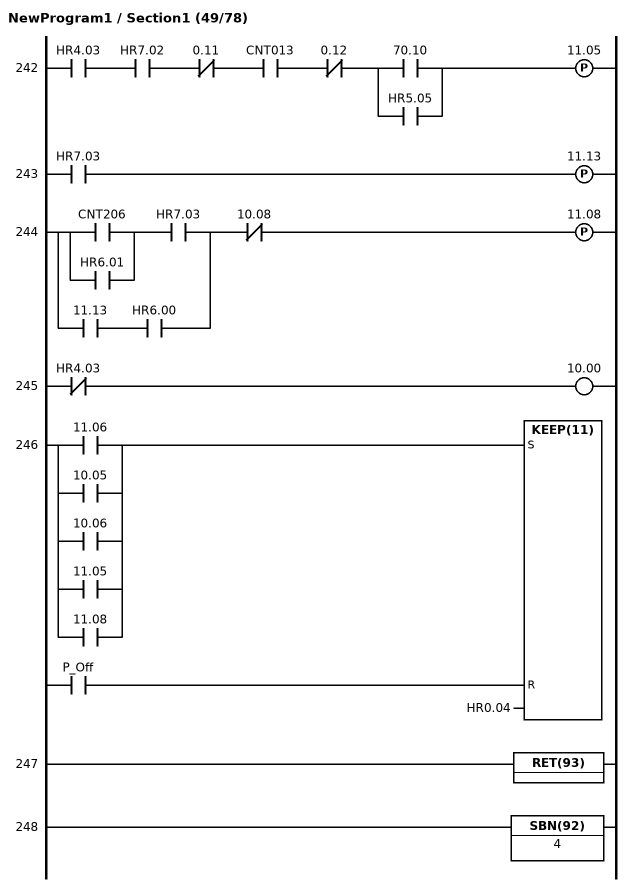
; [picture p48: NewProgram1 / Section1, rungs 242-248]
; rung 242
LD HR4.03
AND HR7.02
ANDNOT 0.11
AND CNT013
ANDNOT 0.12
LD 70.10
OR HR5.05
ANDLD
DIFU(13) 11.05
; rung 243
LD HR7.03
DIFU(13) 11.13
; rung 244
LD CNT206
OR HR6.01
AND HR7.03
LD 11.13
AND HR6.00
ORLD
ANDNOT 10.08
DIFU(13) 11.08
; rung 245
LDNOT HR4.03
OUT 10.00
; rung 246
LD 11.06
OR 10.05
OR 10.06
OR 11.05
OR 11.08
LD P_Off
KEEP(11) HR0.04
; rung 247
RET(93)
; rung 248
SBN(92) 4

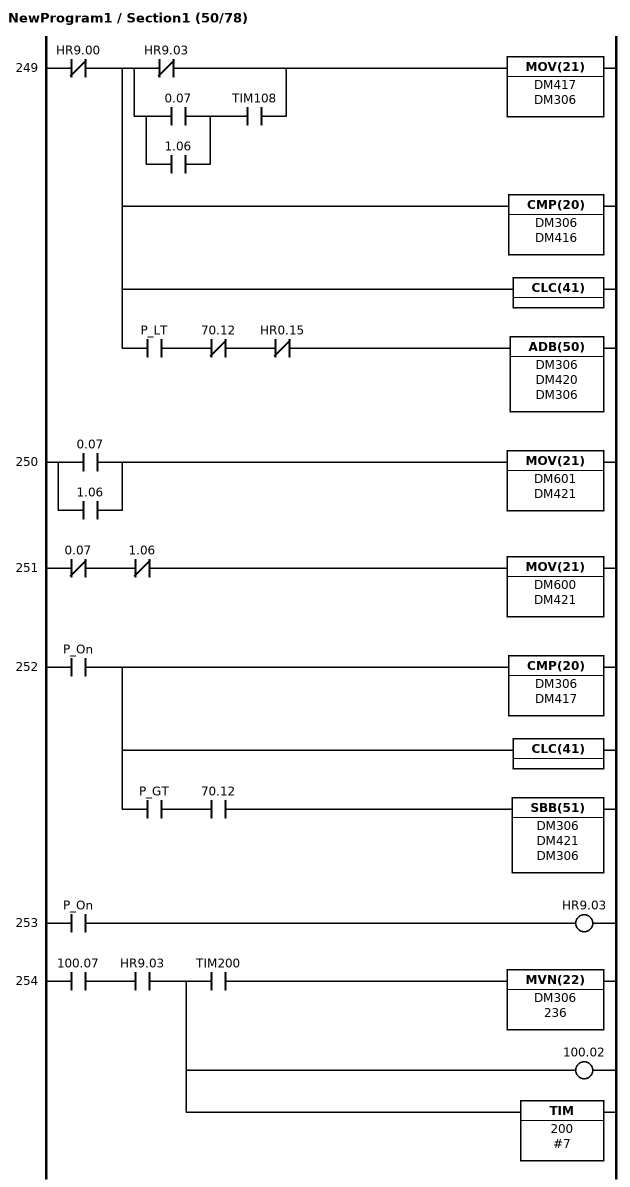
; rung 249
LDNOT HR9.00
OUT TR0
LDNOT HR9.03
LD 0.07
OR 1.06
AND TIM108
ORLD
ANDLD
MOV(21) DM417 DM306
LD TR0
CMP(20) DM306 DM416
CLC(41)
AND P_LT
ANDNOT 70.12
ANDNOT HR0.15
ADB(50) DM306 DM420 DM306
; rung 250
LD 0.07
OR 1.06
MOV(21) DM601 DM421
; rung 251
LDNOT 0.07
ANDNOT 1.06
MOV(21) DM600 DM421
; rung 252
LD P_On
CMP(20) DM306 DM417
CLC(41)
AND P_GT
AND 70.12
SBB(51) DM306 DM421 DM306
; rung 253
LD P_On
OUT HR9.03
; rung 254
LD 100.07
AND HR9.03
OUT TR0
AND TIM200
MVN(22) DM306 236
LD TR0
OUT 100.02
TIM 200 #7

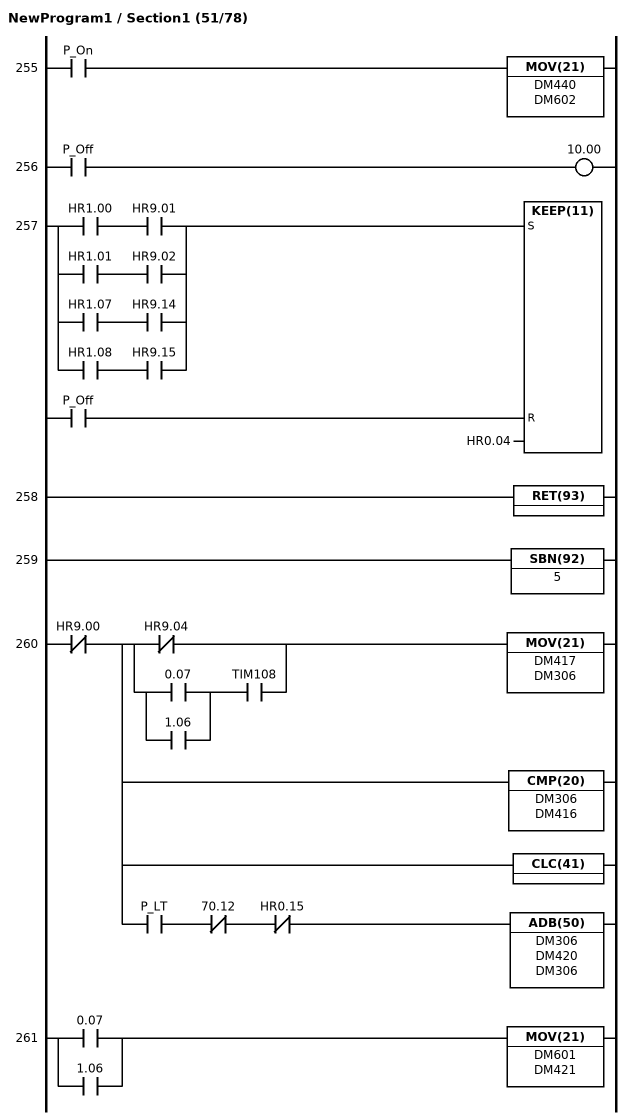
; rung 255
LD P_On
MOV(21) DM440 DM602
; rung 256
LD P_Off
OUT 10.00
; rung 257
LD HR1.00
AND HR9.01
LD HR1.01
AND HR9.02
ORLD
LD HR1.07
AND HR9.14
ORLD
LD HR1.08
AND HR9.15
ORLD
LD P_Off
KEEP(11) HR0.04
; rung 258
RET(93)
; rung 259
SBN(92) 5
; rung 260
LDNOT HR9.00
OUT TR0
LDNOT HR9.04
LD 0.07
OR 1.06
AND TIM108
ORLD
ANDLD
MOV(21) DM417 DM306
LD TR0
CMP(20) DM306 DM416
CLC(41)
AND P_LT
ANDNOT 70.12
ANDNOT HR0.15
ADB(50) DM306 DM420 DM306
; rung 261
LD 0.07
OR 1.06
MOV(21) DM601 DM421

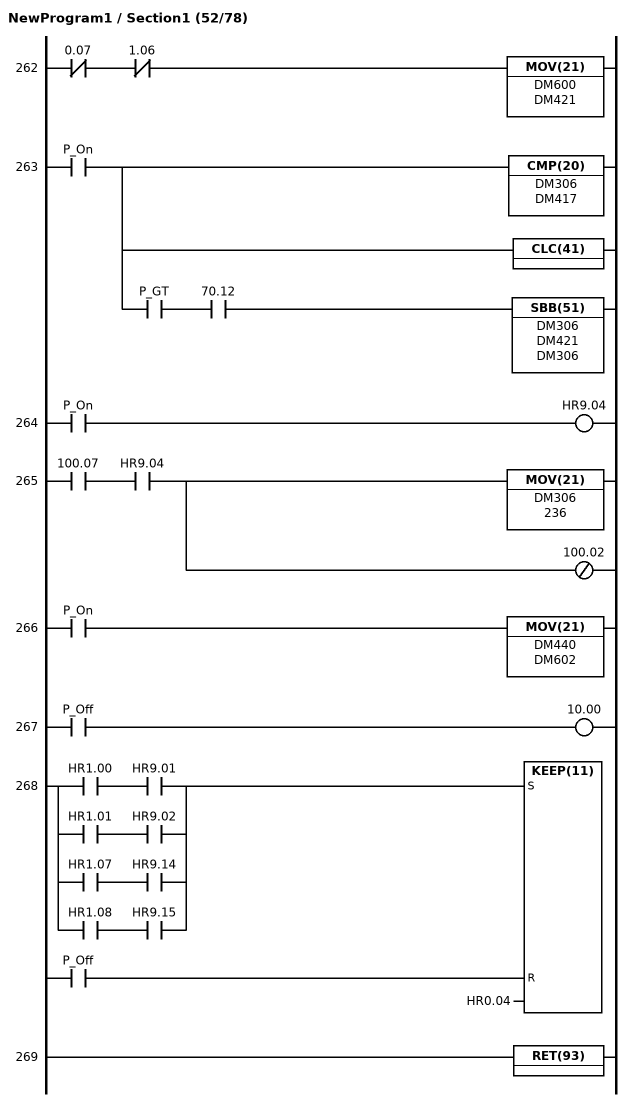
; rung 262
LDNOT 0.07
ANDNOT 1.06
MOV(21) DM600 DM421
; rung 263
LD P_On
CMP(20) DM306 DM417
CLC(41)
AND P_GT
AND 70.12
SBB(51) DM306 DM421 DM306
; rung 264
LD P_On
OUT HR9.04
; rung 265
LD 100.07
AND HR9.04
MOV(21) DM306 236
OUTNOT 100.02
; rung 266
LD P_On
MOV(21) DM440 DM602
; rung 267
LD P_Off
OUT 10.00
; rung 268
LD HR1.00
AND HR9.01
LD HR1.01
AND HR9.02
ORLD
LD HR1.07
AND HR9.14
ORLD
LD HR1.08
AND HR9.15
ORLD
LD P_Off
KEEP(11) HR0.04
; rung 269
RET(93)

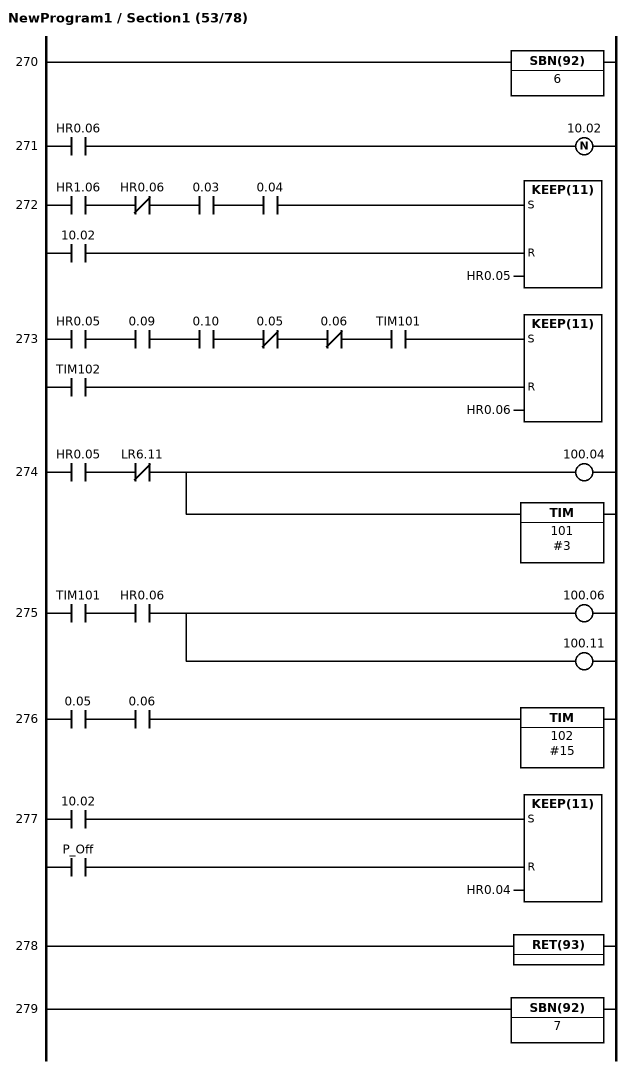
; rung 270
SBN(92) 6
; rung 271
LD HR0.06
DIFD(14) 10.02
; rung 272
LD HR1.06
ANDNOT HR0.06
AND 0.03
AND 0.04
LD 10.02
KEEP(11) HR0.05
; rung 273
LD HR0.05
AND 0.09
AND 0.10
ANDNOT 0.05
ANDNOT 0.06
AND TIM101
LD TIM102
KEEP(11) HR0.06
; rung 274
LD HR0.05
ANDNOT LR6.11
OUT 100.04
TIM 101 #3
; rung 275
LD TIM101
AND HR0.06
OUT 100.06
OUT 100.11
; rung 276
LD 0.05
AND 0.06
TIM 102 #15
; rung 277
LD 10.02
LD P_Off
KEEP(11) HR0.04
; rung 278
RET(93)
; rung 279
SBN(92) 7

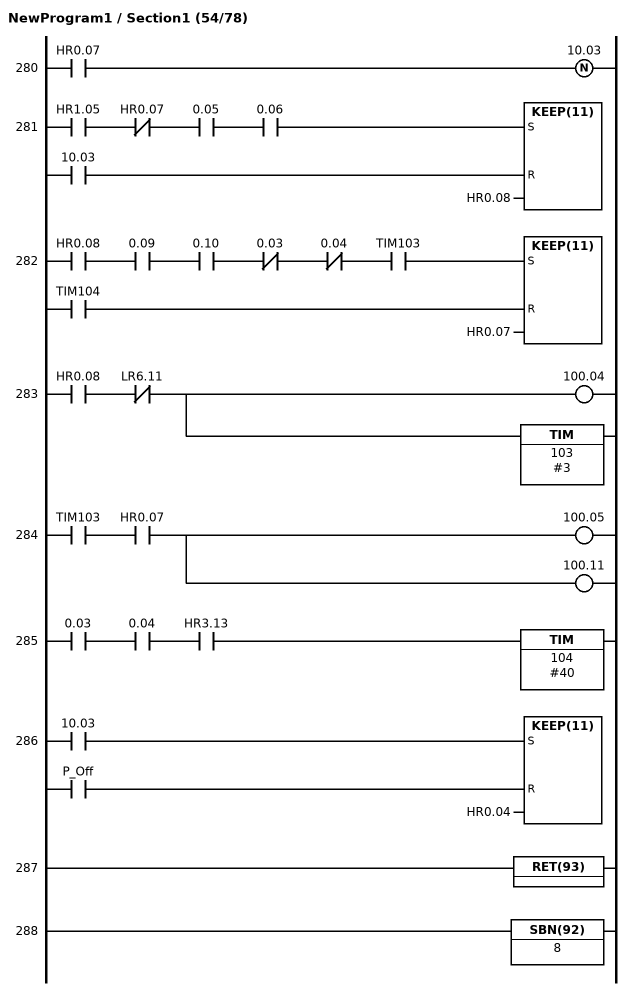
; rung 280
LD HR0.07
DIFD(14) 10.03
; rung 281
LD HR1.05
ANDNOT HR0.07
AND 0.05
AND 0.06
LD 10.03
KEEP(11) HR0.08
; rung 282
LD HR0.08
AND 0.09
AND 0.10
ANDNOT 0.03
ANDNOT 0.04
AND TIM103
LD TIM104
KEEP(11) HR0.07
; rung 283
LD HR0.08
ANDNOT LR6.11
OUT 100.04
TIM 103 #3
; rung 284
LD TIM103
AND HR0.07
OUT 100.05
OUT 100.11
; rung 285
LD 0.03
AND 0.04
AND HR3.13
TIM 104 #40
; rung 286
LD 10.03
LD P_Off
KEEP(11) HR0.04
; rung 287
RET(93)
; rung 288
SBN(92) 8

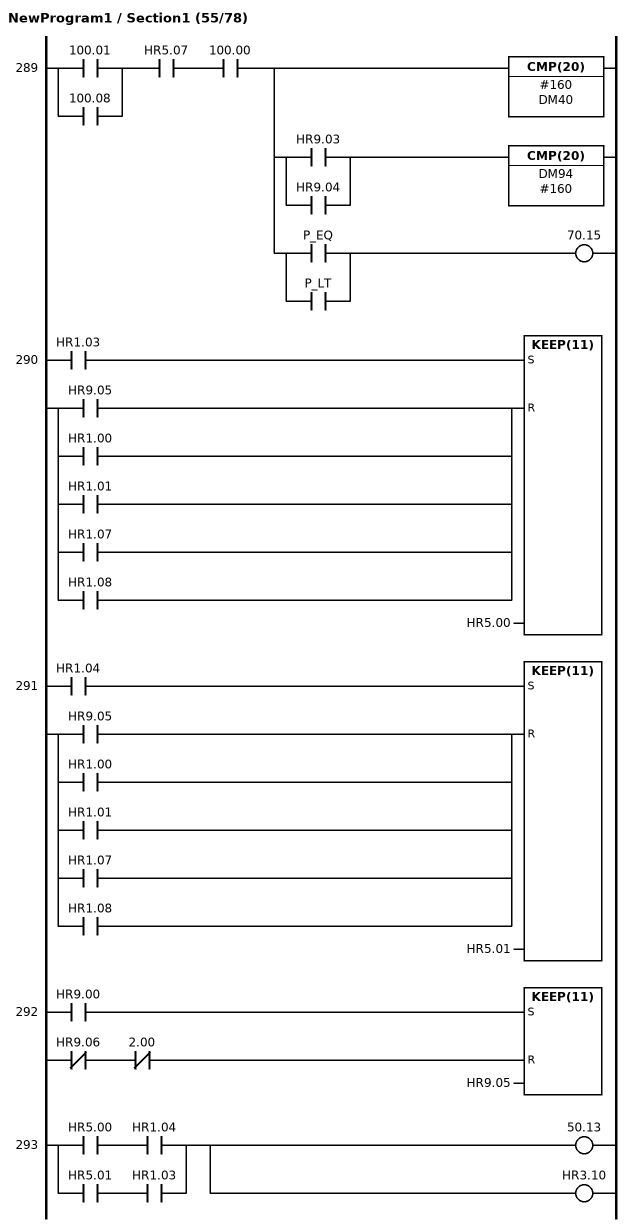
; rung 289
LD 100.01
OR 100.08
AND HR5.07
AND 100.00
OUT TR0
CMP(20) #160 DM40
LD HR9.03
OR HR9.04
ANDLD
CMP(20) DM94 #160
LD TR0
LD P_EQ
OR P_LT
ANDLD
OUT 70.15
; rung 290
LD HR1.03
LD HR9.05
OR HR1.00
OR HR1.01
OR HR1.07
OR HR1.08
KEEP(11) HR5.00
; rung 291
LD HR1.04
LD HR9.05
OR HR1.00
OR HR1.01
OR HR1.07
OR HR1.08
KEEP(11) HR5.01
; rung 292
LD HR9.00
LDNOT HR9.06
ANDNOT 2.00
KEEP(11) HR9.05
; rung 293
LD HR5.00
AND HR1.04
LD HR5.01
AND HR1.03
ORLD
OUT 50.13
OUT HR3.10

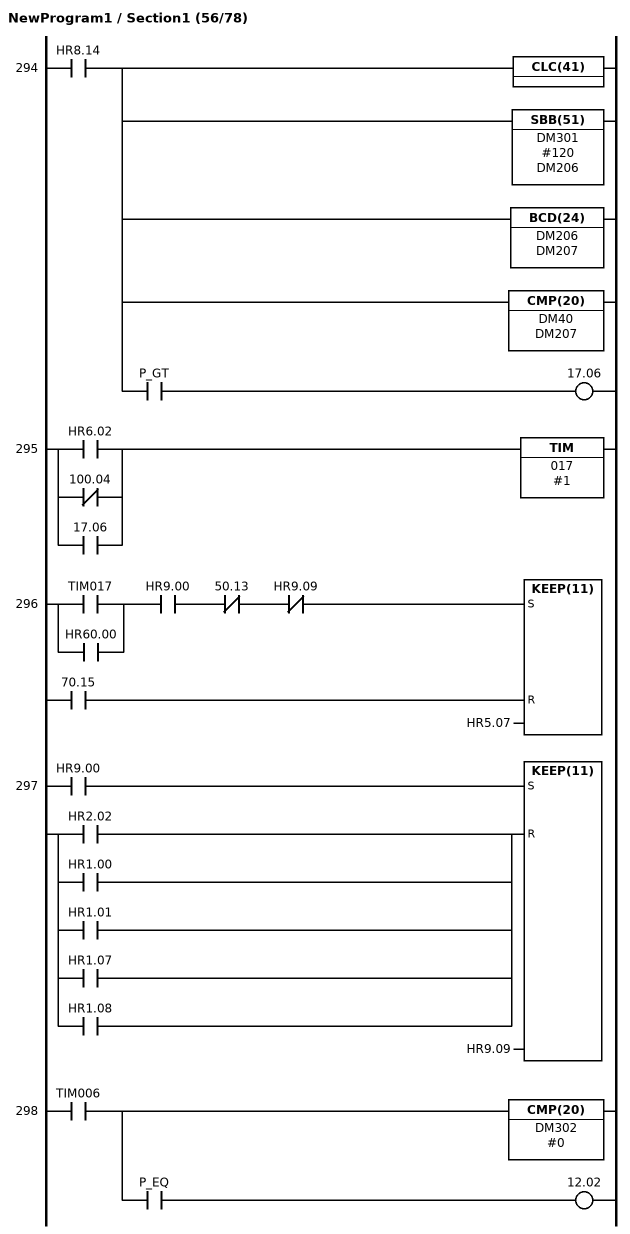
; rung 294
LD HR8.14
CLC(41)
SBB(51) DM301 #120 DM206
BCD(24) DM206 DM207
CMP(20) DM40 DM207
AND P_GT
OUT 17.06
; rung 295
LD HR6.02
ORNOT 100.04
OR 17.06
TIM 017 #1
; rung 296
LD TIM017
OR HR60.00
AND HR9.00
ANDNOT 50.13
ANDNOT HR9.09
LD 70.15
KEEP(11) HR5.07
; rung 297
LD HR9.00
LD HR2.02
OR HR1.00
OR HR1.01
OR HR1.07
OR HR1.08
KEEP(11) HR9.09
; rung 298
LD TIM006
CMP(20) DM302 #0
AND P_EQ
OUT 12.02

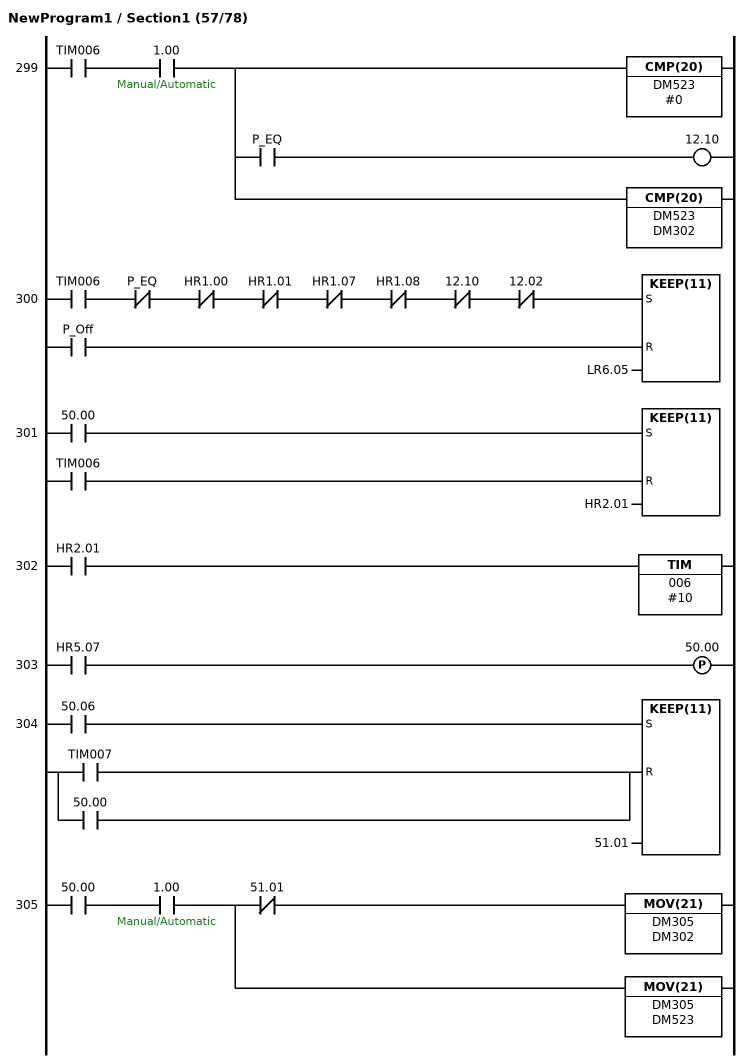
; rung 299
LD TIM006
AND 1.00  ; Manual/Automatic
OUT TR0
CMP(20) DM523 #0
AND P_EQ
OUT 12.10
LD TR0
CMP(20) DM523 DM302
; rung 300
LD TIM006
ANDNOT P_EQ
ANDNOT HR1.00
ANDNOT HR1.01
ANDNOT HR1.07
ANDNOT HR1.08
ANDNOT 12.10
ANDNOT 12.02
LD P_Off
KEEP(11) LR6.05
; rung 301
LD 50.00
LD TIM006
KEEP(11) HR2.01
; rung 302
LD HR2.01
TIM 006 #10
; rung 303
LD HR5.07
DIFU(13) 50.00
; rung 304
LD 50.06
LD TIM007
OR 50.00
KEEP(11) 51.01
; rung 305
LD 50.00
AND 1.00  ; Manual/Automatic
OUT TR0
ANDNOT 51.01
MOV(21) DM305 DM302
LD TR0
MOV(21) DM305 DM523

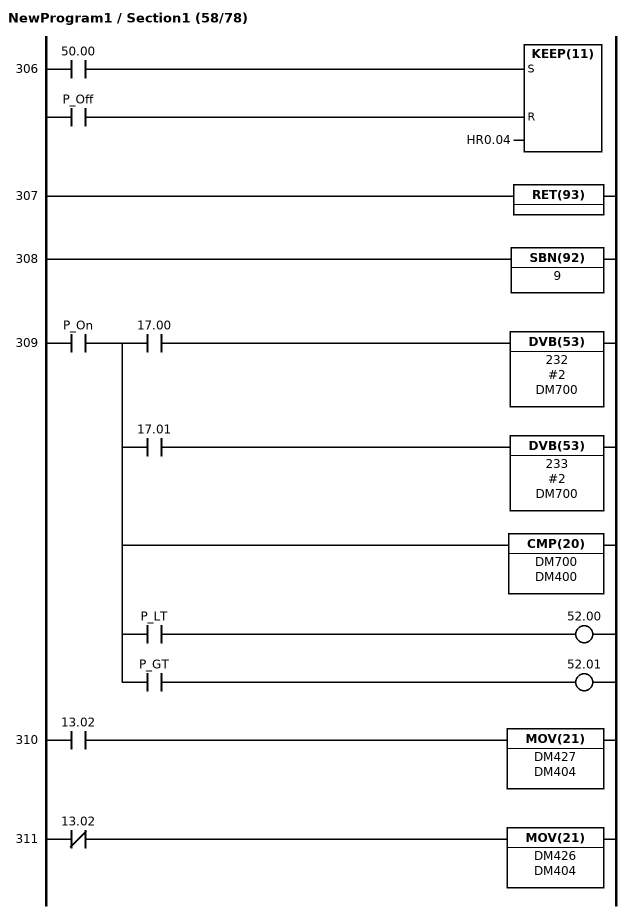
; rung 306
LD 50.00
LD P_Off
KEEP(11) HR0.04
; rung 307
RET(93)
; rung 308
SBN(92) 9
; rung 309
LD P_On
OUT TR0
AND 17.00
DVB(53) 232 #2 DM700
LD TR0
AND 17.01
DVB(53) 233 #2 DM700
LD TR0
CMP(20) DM700 DM400
AND P_LT
OUT 52.00
LD TR0
AND P_GT
OUT 52.01
; rung 310
LD 13.02
MOV(21) DM427 DM404
; rung 311
LDNOT 13.02
MOV(21) DM426 DM404

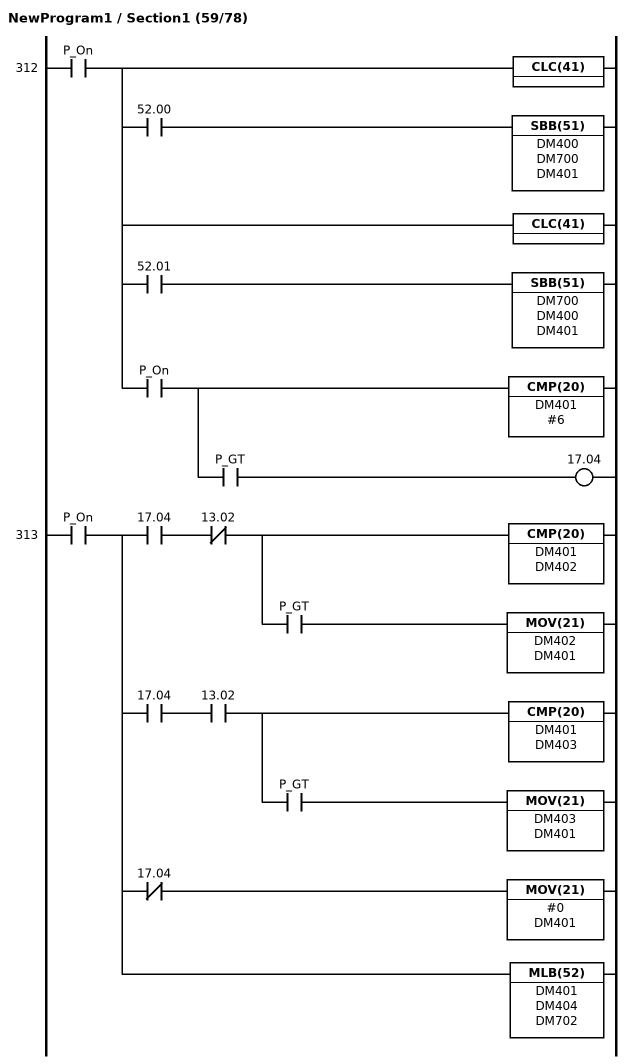
; rung 312
LD P_On
OUT TR0
CLC(41)
AND 52.00
SBB(51) DM400 DM700 DM401
LD TR0
CLC(41)
AND 52.01
SBB(51) DM700 DM400 DM401
LD TR0
AND P_On
CMP(20) DM401 #6
AND P_GT
OUT 17.04
; rung 313
LD P_On
OUT TR0
AND 17.04
ANDNOT 13.02
CMP(20) DM401 DM402
AND P_GT
MOV(21) DM402 DM401
LD TR0
AND 17.04
AND 13.02
CMP(20) DM401 DM403
AND P_GT
MOV(21) DM403 DM401
LD TR0
ANDNOT 17.04
MOV(21) #0 DM401
LD TR0
MLB(52) DM401 DM404 DM702

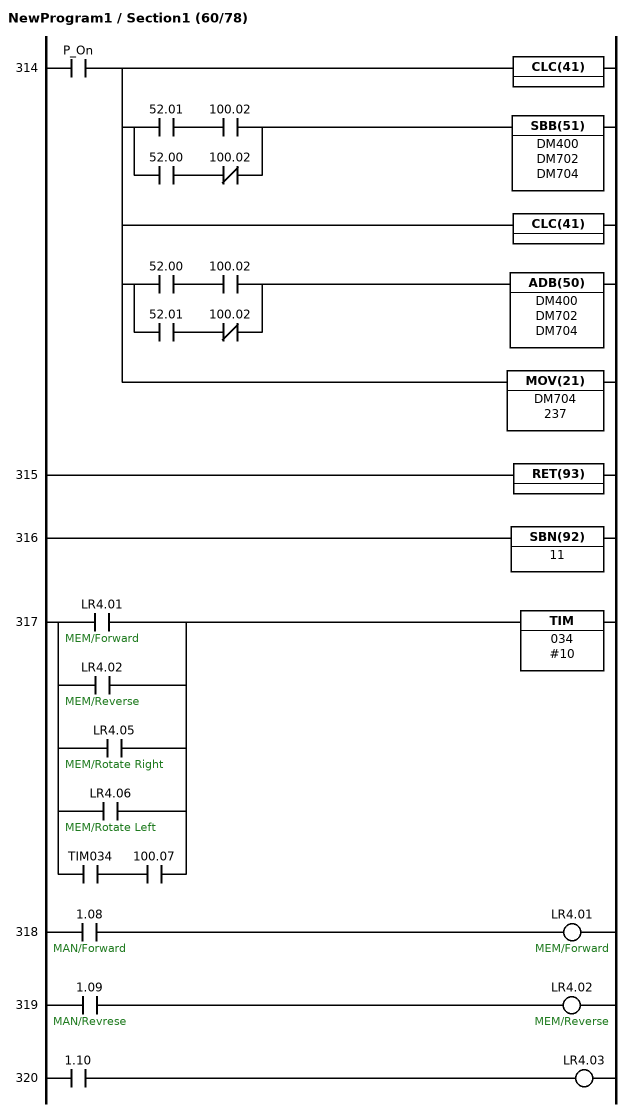
; rung 314
LD P_On
OUT TR0
CLC(41)
LD 52.01
AND 100.02
LD 52.00
ANDNOT 100.02
ORLD
ANDLD
SBB(51) DM400 DM702 DM704
LD TR0
CLC(41)
LD 52.00
AND 100.02
LD 52.01
ANDNOT 100.02
ORLD
ANDLD
ADB(50) DM400 DM702 DM704
LD TR0
MOV(21) DM704 237
; rung 315
RET(93)
; rung 316
SBN(92) 11
; rung 317
LD LR4.01  ; MEM/Forward
OR LR4.02  ; MEM/Reverse
OR LR4.05  ; MEM/Rotate Right
OR LR4.06  ; MEM/Rotate Left
LD TIM034
AND 100.07
ORLD
TIM 034 #10
; rung 318
LD 1.08  ; MAN/Forward
OUT LR4.01  ; MEM/Forward
; rung 319
LD 1.09  ; MAN/Revrese
OUT LR4.02  ; MEM/Reverse
; rung 320
LD 1.10
OUT LR4.03

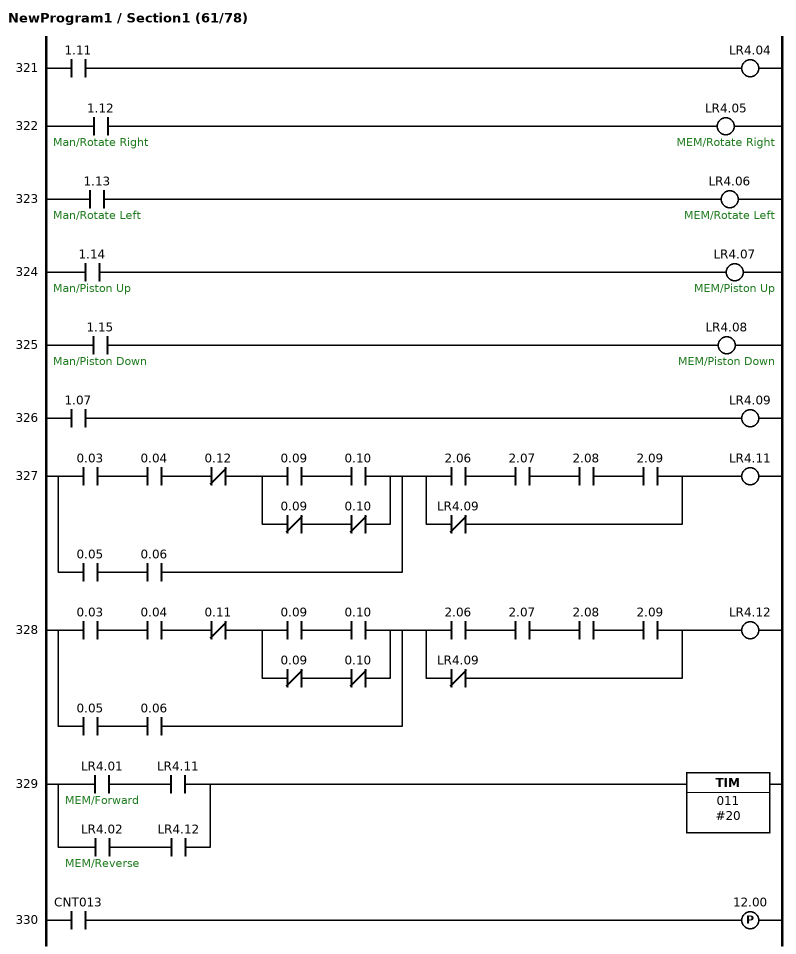
; rung 321
LD 1.11
OUT LR4.04
; rung 322
LD 1.12  ; Man/Rotate Right
OUT LR4.05  ; MEM/Rotate Right
; rung 323
LD 1.13  ; Man/Rotate Left
OUT LR4.06  ; MEM/Rotate Left
; rung 324
LD 1.14  ; Man/Piston Up
OUT LR4.07  ; MEM/Piston Up
; rung 325
LD 1.15  ; Man/Piston Down
OUT LR4.08  ; MEM/Piston Down
; rung 326
LD 1.07
OUT LR4.09
; rung 327
LD 0.03
AND 0.04
ANDNOT 0.12
LD 0.09
AND 0.10
LDNOT 0.09
ANDNOT 0.10
ORLD
ANDLD
LD 0.05
AND 0.06
ORLD
LD 2.06
AND 2.07
AND 2.08
AND 2.09
ORNOT LR4.09
ANDLD
OUT LR4.11
; rung 328
LD 0.03
AND 0.04
ANDNOT 0.11
LD 0.09
AND 0.10
LDNOT 0.09
ANDNOT 0.10
ORLD
ANDLD
LD 0.05
AND 0.06
ORLD
LD 2.06
AND 2.07
AND 2.08
AND 2.09
ORNOT LR4.09
ANDLD
OUT LR4.12
; rung 329
LD LR4.01  ; MEM/Forward
AND LR4.11
LD LR4.02  ; MEM/Reverse
AND LR4.12
ORLD
TIM 011 #20
; rung 330
LD CNT013
DIFU(13) 12.00

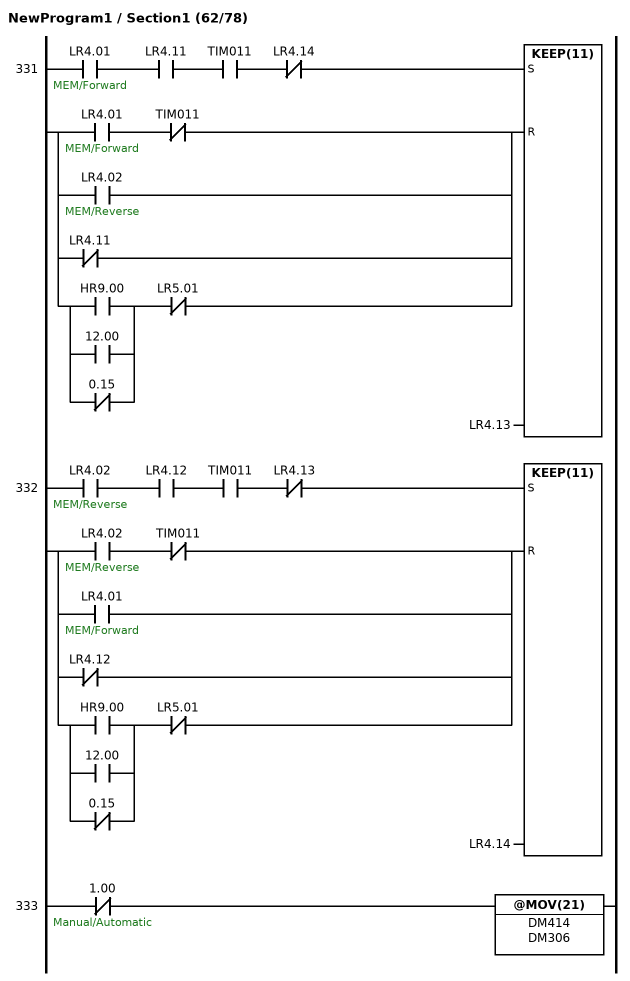
; rung 331
LD LR4.01  ; MEM/Forward
AND LR4.11
AND TIM011
ANDNOT LR4.14
LD LR4.01  ; MEM/Forward
ANDNOT TIM011
OR LR4.02  ; MEM/Reverse
ORNOT LR4.11
LD HR9.00
OR 12.00
ORNOT 0.15
ANDNOT LR5.01
ORLD
KEEP(11) LR4.13
; rung 332
LD LR4.02  ; MEM/Reverse
AND LR4.12
AND TIM011
ANDNOT LR4.13
LD LR4.02  ; MEM/Reverse
ANDNOT TIM011
OR LR4.01  ; MEM/Forward
ORNOT LR4.12
LD HR9.00
OR 12.00
ORNOT 0.15
ANDNOT LR5.01
ORLD
KEEP(11) LR4.14
; rung 333
LDNOT 1.00  ; Manual/Automatic
@MOV(21) DM414 DM306

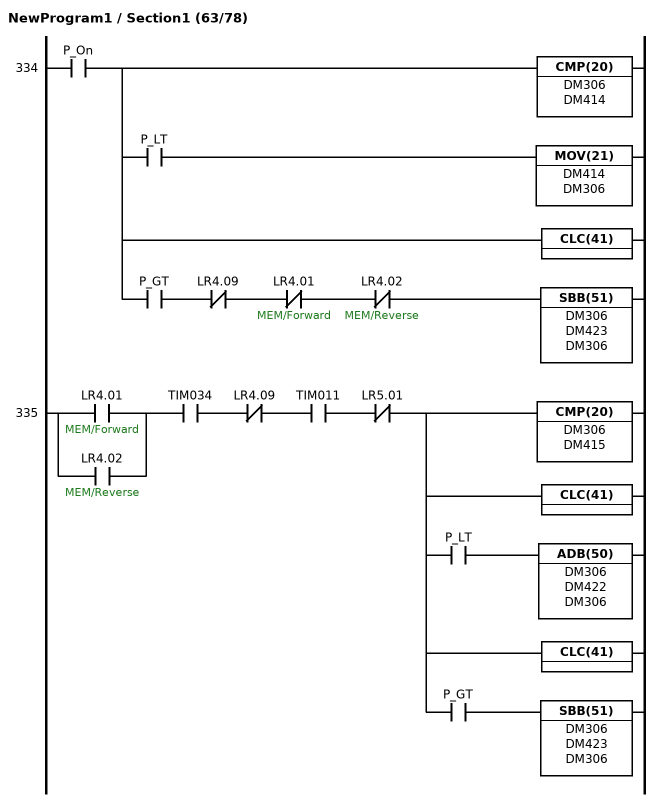
; rung 334
LD P_On
OUT TR0
CMP(20) DM306 DM414
AND P_LT
MOV(21) DM414 DM306
LD TR0
CLC(41)
AND P_GT
ANDNOT LR4.09
ANDNOT LR4.01  ; MEM/Forward
ANDNOT LR4.02  ; MEM/Reverse
SBB(51) DM306 DM423 DM306
; rung 335
LD LR4.01  ; MEM/Forward
OR LR4.02  ; MEM/Reverse
AND TIM034
ANDNOT LR4.09
AND TIM011
ANDNOT LR5.01
OUT TR0
CMP(20) DM306 DM415
CLC(41)
AND P_LT
ADB(50) DM306 DM422 DM306
LD TR0
CLC(41)
AND P_GT
SBB(51) DM306 DM423 DM306

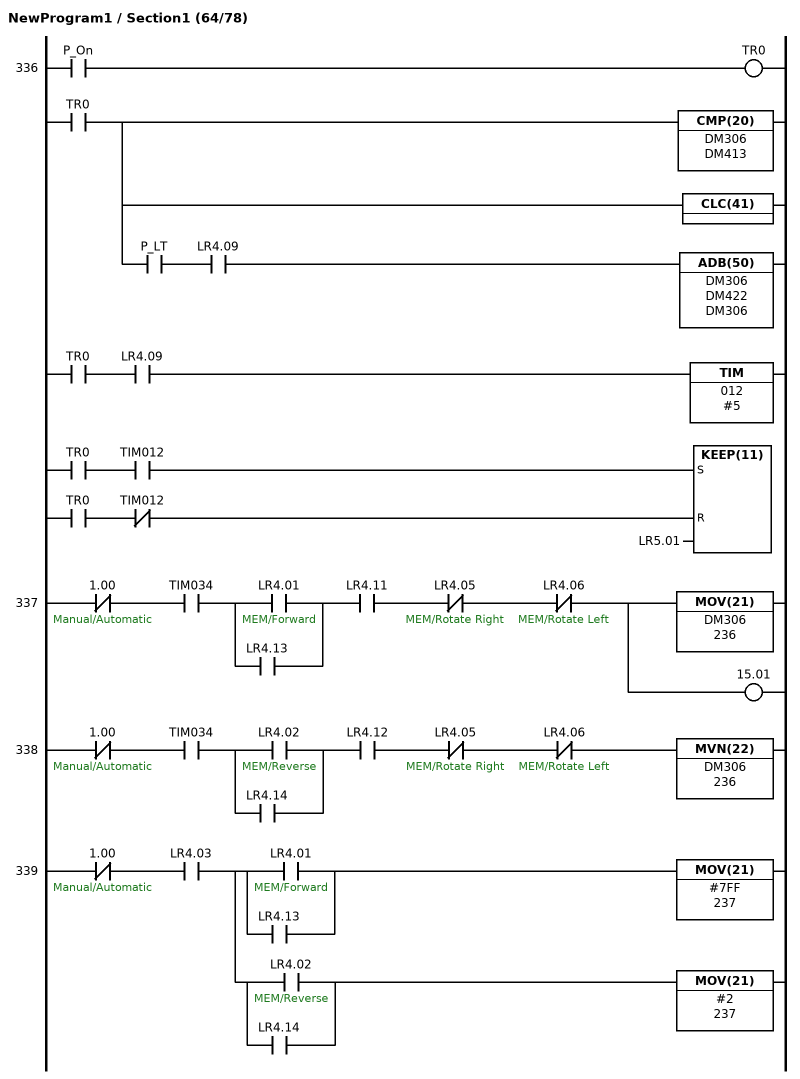
; rung 336
LD P_On
OUT TR0
CMP(20) DM306 DM413
CLC(41)
AND P_LT
AND LR4.09
ADB(50) DM306 DM422 DM306
LD TR0
AND LR4.09
TIM 012 #5
LD TR0
AND TIM012
LD TR0
ANDNOT TIM012
KEEP(11) LR5.01
; rung 337
LDNOT 1.00  ; Manual/Automatic
AND TIM034
LD LR4.01  ; MEM/Forward
OR LR4.13
ANDLD
AND LR4.11
ANDNOT LR4.05  ; MEM/Rotate Right
ANDNOT LR4.06  ; MEM/Rotate Left
MOV(21) DM306 236
OUT 15.01
; rung 338
LDNOT 1.00  ; Manual/Automatic
AND TIM034
LD LR4.02  ; MEM/Reverse
OR LR4.14
ANDLD
AND LR4.12
ANDNOT LR4.05  ; MEM/Rotate Right
ANDNOT LR4.06  ; MEM/Rotate Left
MVN(22) DM306 236
; rung 339
LDNOT 1.00  ; Manual/Automatic
AND LR4.03
OUT TR0
LD LR4.01  ; MEM/Forward
OR LR4.13
ANDLD
MOV(21) #7FF 237
LD TR0
LD LR4.02  ; MEM/Reverse
OR LR4.14
ANDLD
MOV(21) #2 237

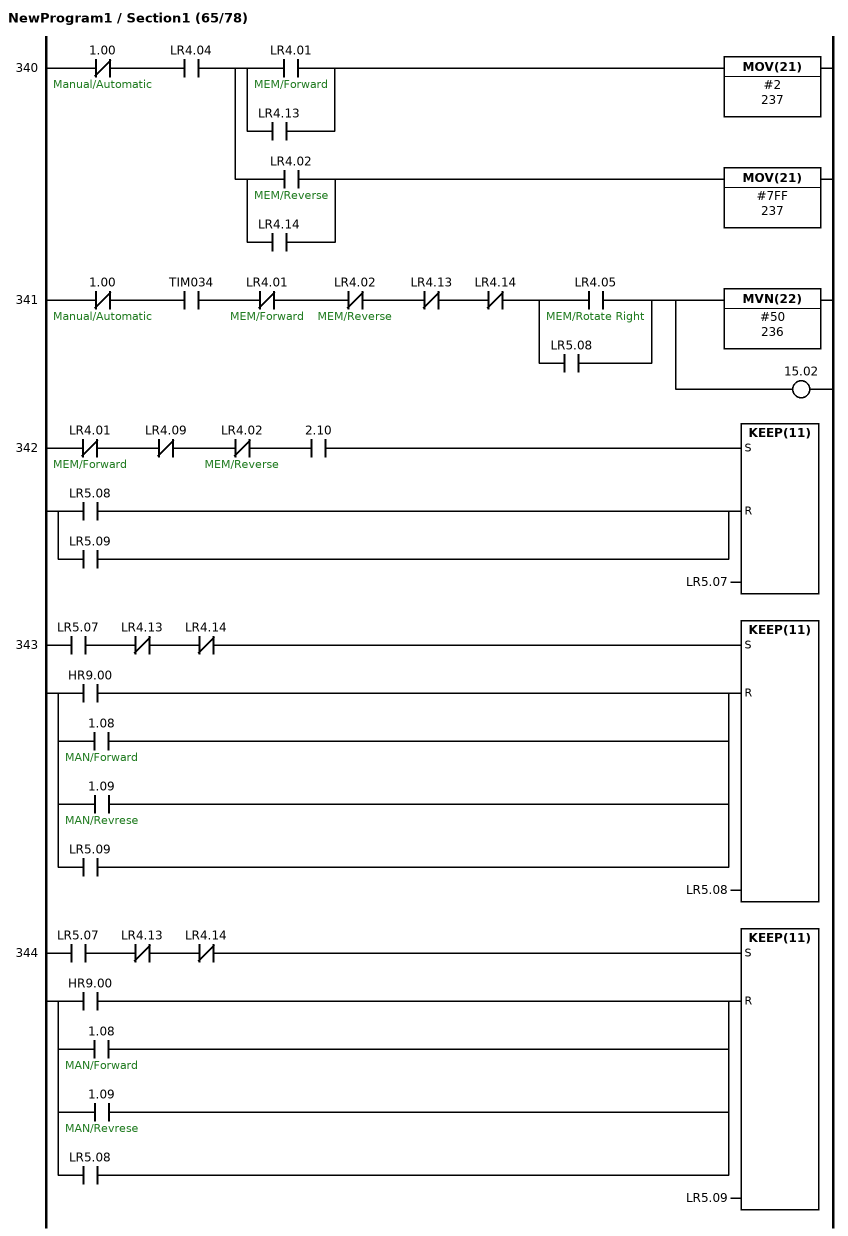
; rung 340
LDNOT 1.00  ; Manual/Automatic
AND LR4.04
OUT TR0
LD LR4.01  ; MEM/Forward
OR LR4.13
ANDLD
MOV(21) #2 237
LD TR0
LD LR4.02  ; MEM/Reverse
OR LR4.14
ANDLD
MOV(21) #7FF 237
; rung 341
LDNOT 1.00  ; Manual/Automatic
AND TIM034
ANDNOT LR4.01  ; MEM/Forward
ANDNOT LR4.02  ; MEM/Reverse
ANDNOT LR4.13
ANDNOT LR4.14
LD LR4.05  ; MEM/Rotate Right
OR LR5.08
ANDLD
MVN(22) #50 236
OUT 15.02
; rung 342
LDNOT LR4.01  ; MEM/Forward
ANDNOT LR4.09
ANDNOT LR4.02  ; MEM/Reverse
AND 2.10
LD LR5.08
OR LR5.09
KEEP(11) LR5.07
; rung 343
LD LR5.07
ANDNOT LR4.13
ANDNOT LR4.14
LD HR9.00
OR 1.08  ; MAN/Forward
OR 1.09  ; MAN/Revrese
OR LR5.09
KEEP(11) LR5.08
; rung 344
LD LR5.07
ANDNOT LR4.13
ANDNOT LR4.14
LD HR9.00
OR 1.08  ; MAN/Forward
OR 1.09  ; MAN/Revrese
OR LR5.08
KEEP(11) LR5.09

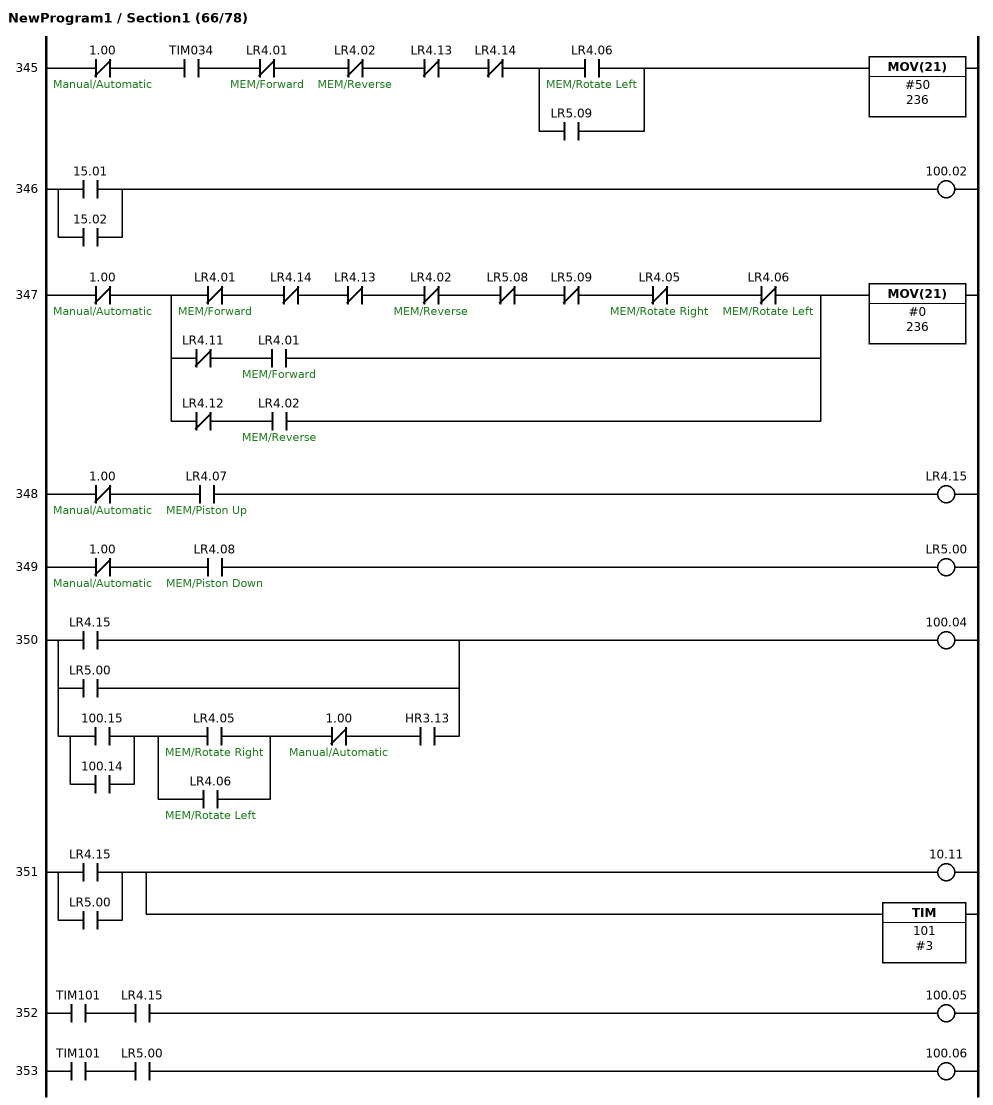
; rung 345
LDNOT 1.00  ; Manual/Automatic
AND TIM034
ANDNOT LR4.01  ; MEM/Forward
ANDNOT LR4.02  ; MEM/Reverse
ANDNOT LR4.13
ANDNOT LR4.14
LD LR4.06  ; MEM/Rotate Left
OR LR5.09
ANDLD
MOV(21) #50 236
; rung 346
LD 15.01
OR 15.02
OUT 100.02
; rung 347
LDNOT 1.00  ; Manual/Automatic
LDNOT LR4.01  ; MEM/Forward
ANDNOT LR4.14
ANDNOT LR4.13
ANDNOT LR4.02  ; MEM/Reverse
ANDNOT LR5.08
ANDNOT LR5.09
ANDNOT LR4.05  ; MEM/Rotate Right
ANDNOT LR4.06  ; MEM/Rotate Left
LDNOT LR4.11
AND LR4.01  ; MEM/Forward
ORLD
LDNOT LR4.12
AND LR4.02  ; MEM/Reverse
ORLD
ANDLD
MOV(21) #0 236
; rung 348
LDNOT 1.00  ; Manual/Automatic
AND LR4.07  ; MEM/Piston Up
OUT LR4.15
; rung 349
LDNOT 1.00  ; Manual/Automatic
AND LR4.08  ; MEM/Piston Down
OUT LR5.00
; rung 350
LD LR4.15
OR LR5.00
LD 100.15
OR 100.14
LD LR4.05  ; MEM/Rotate Right
OR LR4.06  ; MEM/Rotate Left
ANDLD
ANDNOT 1.00  ; Manual/Automatic
AND HR3.13
ORLD
OUT 100.04
; rung 351
LD LR4.15
OR LR5.00
OUT 10.11
TIM 101 #3
; rung 352
LD TIM101
AND LR4.15
OUT 100.05
; rung 353
LD TIM101
AND LR5.00
OUT 100.06

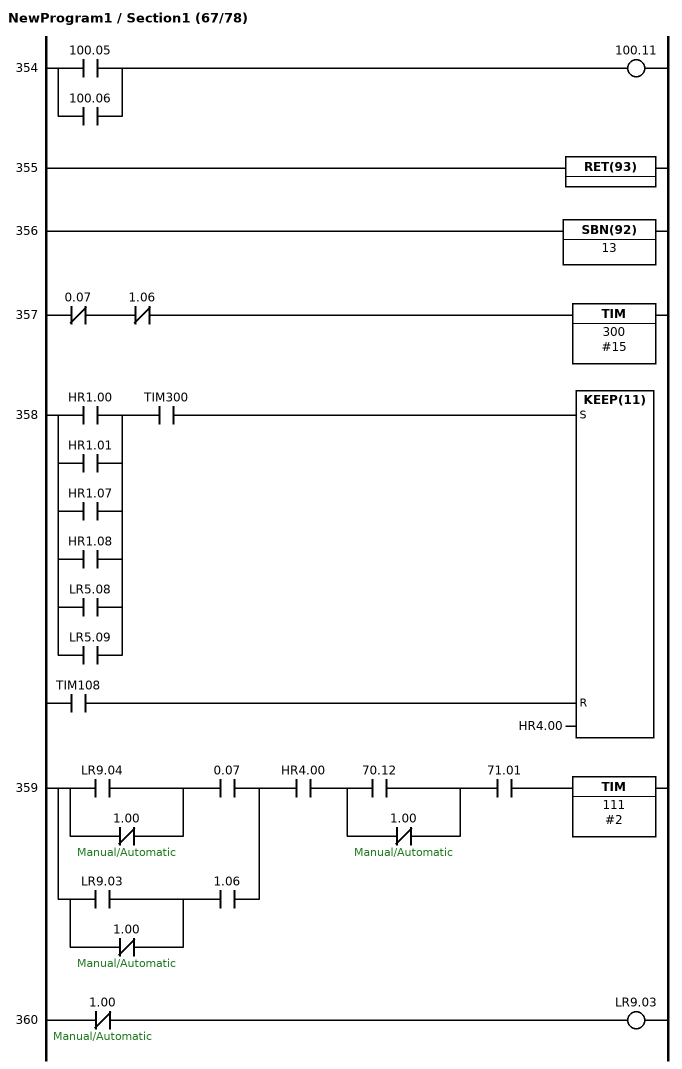
; rung 354
LD 100.05
OR 100.06
OUT 100.11
; rung 355
RET(93)
; rung 356
SBN(92) 13
; rung 357
LDNOT 0.07
ANDNOT 1.06
TIM 300 #15
; rung 358
LD HR1.00
OR HR1.01
OR HR1.07
OR HR1.08
OR LR5.08
OR LR5.09
AND TIM300
LD TIM108
KEEP(11) HR4.00
; rung 359
LD LR9.04
ORNOT 1.00  ; Manual/Automatic
AND 0.07
LD LR9.03
ORNOT 1.00  ; Manual/Automatic
AND 1.06
ORLD
AND HR4.00
LD 70.12
ORNOT 1.00  ; Manual/Automatic
ANDLD
AND 71.01
TIM 111 #2
; rung 360
LDNOT 1.00  ; Manual/Automatic
OUT LR9.03

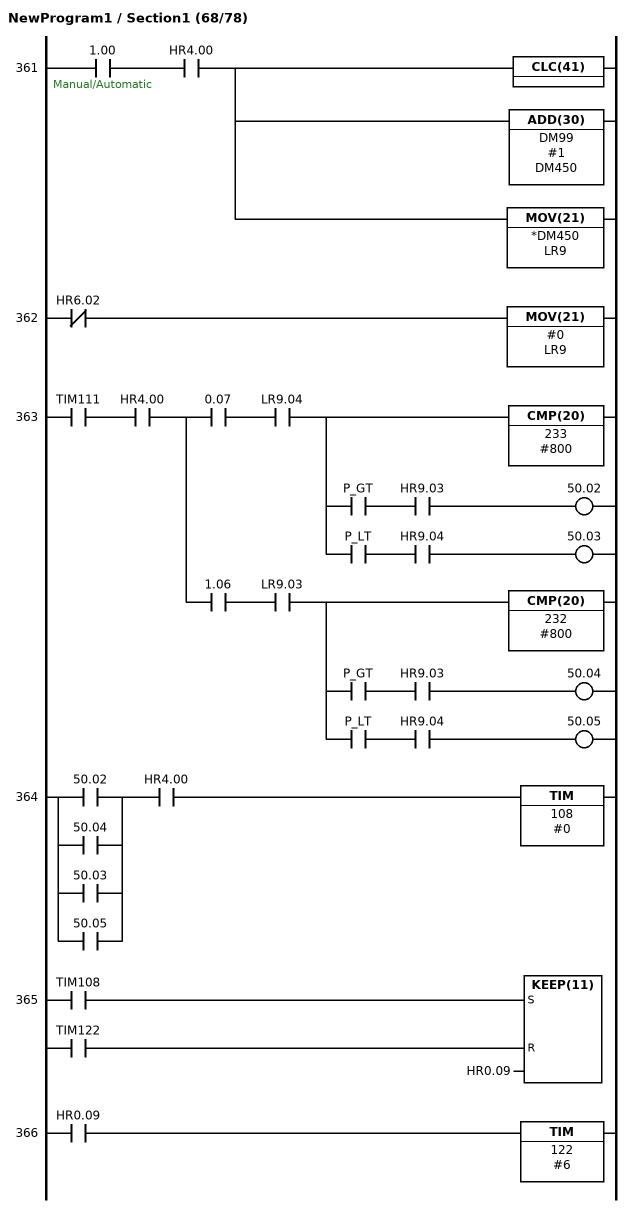
; rung 361
LD 1.00  ; Manual/Automatic
AND HR4.00
CLC(41)
ADD(30) DM99 #1 DM450
MOV(21) *DM450 LR9
; rung 362
LDNOT HR6.02
MOV(21) #0 LR9
; rung 363
LD TIM111
AND HR4.00
OUT TR0
AND 0.07
AND LR9.04
OUT TR1
CMP(20) 233 #800
AND P_GT
AND HR9.03
OUT 50.02
LD TR1
AND P_LT
AND HR9.04
OUT 50.03
LD TR0
AND 1.06
AND LR9.03
OUT TR0
CMP(20) 232 #800
AND P_GT
AND HR9.03
OUT 50.04
LD TR0
AND P_LT
AND HR9.04
OUT 50.05
; rung 364
LD 50.02
OR 50.04
OR 50.03
OR 50.05
AND HR4.00
TIM 108 #0
; rung 365
LD TIM108
LD TIM122
KEEP(11) HR0.09
; rung 366
LD HR0.09
TIM 122 #6

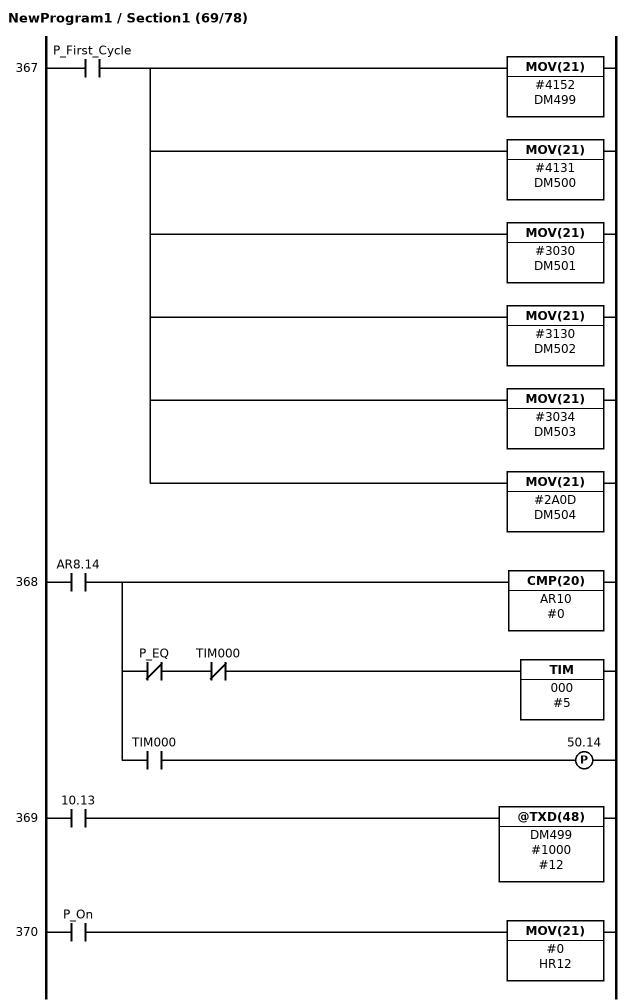
; rung 367
LD P_First_Cycle
MOV(21) #4152 DM499
MOV(21) #4131 DM500
MOV(21) #3030 DM501
MOV(21) #3130 DM502
MOV(21) #3034 DM503
MOV(21) #2A0D DM504
; rung 368
LD AR8.14
OUT TR0
CMP(20) AR10 #0
ANDNOT P_EQ
ANDNOT TIM000
TIM 000 #5
LD TR0
AND TIM000
DIFU(13) 50.14
; rung 369
LD 10.13
@TXD(48) DM499 #1000 #12
; rung 370
LD P_On
MOV(21) #0 HR12

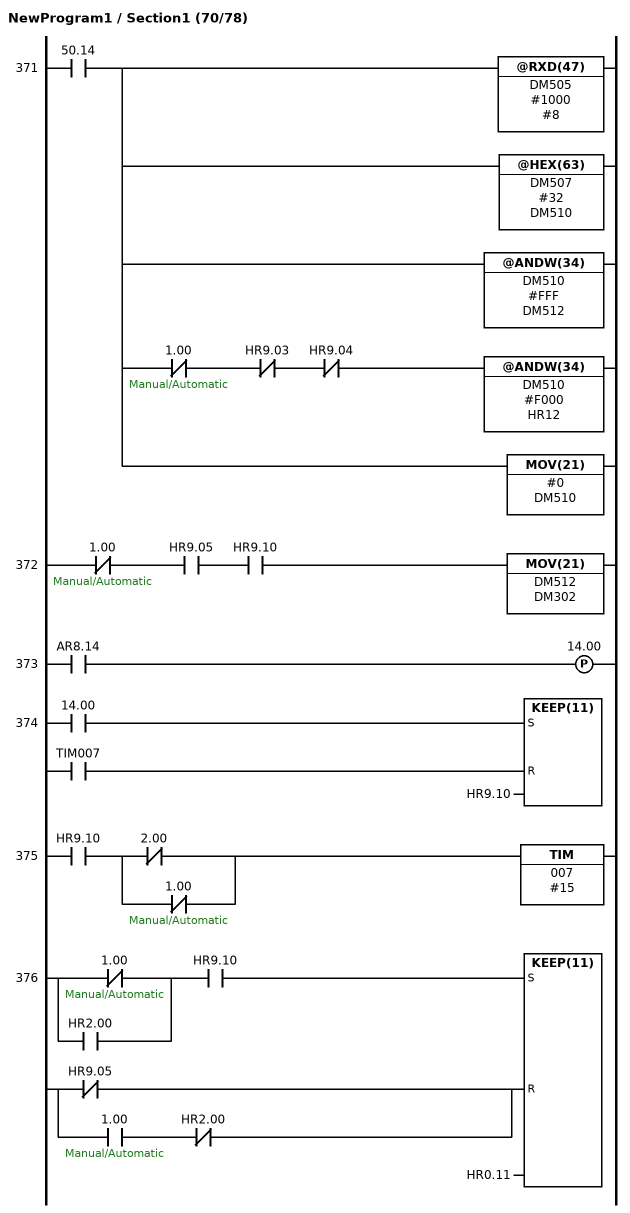
; rung 371
LD 50.14
OUT TR0
@RXD(47) DM505 #1000 #8
@HEX(63) DM507 #32 DM510
@ANDW(34) DM510 #FFF DM512
ANDNOT 1.00  ; Manual/Automatic
ANDNOT HR9.03
ANDNOT HR9.04
@ANDW(34) DM510 #F000 HR12
LD TR0
MOV(21) #0 DM510
; rung 372
LDNOT 1.00  ; Manual/Automatic
AND HR9.05
AND HR9.10
MOV(21) DM512 DM302
; rung 373
LD AR8.14
DIFU(13) 14.00
; rung 374
LD 14.00
LD TIM007
KEEP(11) HR9.10
; rung 375
LD HR9.10
LDNOT 2.00
ORNOT 1.00  ; Manual/Automatic
ANDLD
TIM 007 #15
; rung 376
LDNOT 1.00  ; Manual/Automatic
OR HR2.00
AND HR9.10
LDNOT HR9.05
LD 1.00  ; Manual/Automatic
ANDNOT HR2.00
ORLD
KEEP(11) HR0.11

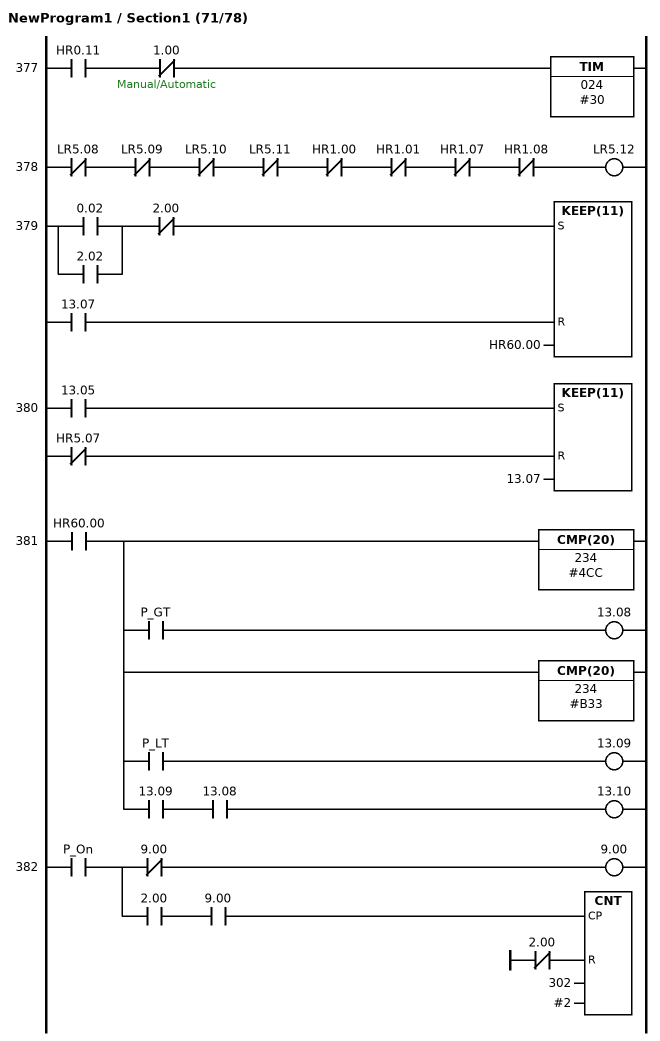
; rung 377
LD HR0.11
ANDNOT 1.00  ; Manual/Automatic
TIM 024 #30
; rung 378
LDNOT LR5.08
ANDNOT LR5.09
ANDNOT LR5.10
ANDNOT LR5.11
ANDNOT HR1.00
ANDNOT HR1.01
ANDNOT HR1.07
ANDNOT HR1.08
OUT LR5.12
; rung 379
LD 0.02
OR 2.02
ANDNOT 2.00
LD 13.07
KEEP(11) HR60.00
; rung 380
LD 13.05
LDNOT HR5.07
KEEP(11) 13.07
; rung 381
LD HR60.00
OUT TR0
CMP(20) 234 #4CC
AND P_GT
OUT 13.08
LD TR0
CMP(20) 234 #B33
AND P_LT
OUT 13.09
LD TR0
AND 13.09
AND 13.08
OUT 13.10
; rung 382
LD P_On
OUT TR0
ANDNOT 9.00
OUT 9.00
LD TR0
AND 2.00
AND 9.00
LDNOT 2.00
CNT 302 #2

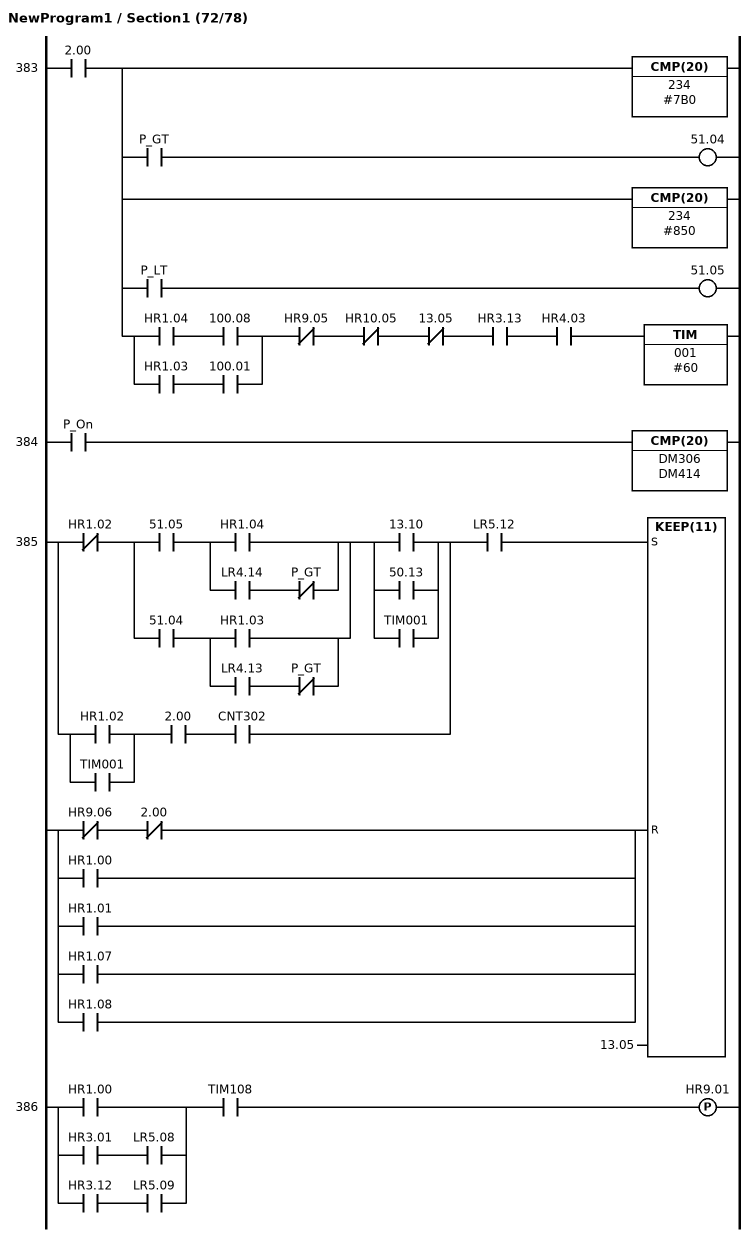
; rung 383
LD 2.00
OUT TR0
CMP(20) 234 #7B0
AND P_GT
OUT 51.04
LD TR0
CMP(20) 234 #850
AND P_LT
OUT 51.05
LD TR0
LD HR1.04
AND 100.08
LD HR1.03
AND 100.01
ORLD
ANDLD
ANDNOT HR9.05
ANDNOT HR10.05
ANDNOT 13.05
AND HR3.13
AND HR4.03
TIM 001 #60
; rung 384
LD P_On
CMP(20) DM306 DM414
; rung 385
LDNOT HR1.02
LD 51.05
LD HR1.04
LD LR4.14
ANDNOT P_GT
ORLD
ANDLD
LD 51.04
LD HR1.03
LD LR4.13
ANDNOT P_GT
ORLD
ANDLD
ORLD
ANDLD
LD 13.10
OR 50.13
OR TIM001
ANDLD
LD HR1.02
OR TIM001
AND 2.00
AND CNT302
ORLD
AND LR5.12
LDNOT HR9.06
ANDNOT 2.00
OR HR1.00
OR HR1.01
OR HR1.07
OR HR1.08
KEEP(11) 13.05
; rung 386
LD HR1.00
LD HR3.01
AND LR5.08
ORLD
LD HR3.12
AND LR5.09
ORLD
AND TIM108
DIFU(13) HR9.01

